PROGRAM WateringTask
VAR
	WaterTimer: TON;
state : INT	 :=0; 	
Delay: Ton;
END_VAR

 	
//Watering control
CASE state OF
	
END_CASE
0:// Initial position
WaterON:= FALSE;
state:=1;
1:// Checking the conditions
IF WaterRequired THEN
            WaterDuration := GetWaterDuration(Moisture, Temp);
            WaterOn := TRUE;
            WaterTimer(IN := TRUE, PT := WaterDuration);
            nState := 2;
        ELSE
            nState := 3;
        END_IF;
		
2:  // Watering
WaterTimer(IN := TRUE);
        IF WaterTimer.Q THEN
          WaterON := FALSE;
WaterRequired := FALSE;
WaterTimer(IN := FALSE);
            state := 3;
3:// Idle
Delay(IN:=TRUE, PT:=T#5S);
IF NOT(Delay.Q) THEN
	RETURN;
END_IF
Delay(In:=FALSE);
state:=1;		
END_CASE

END_PROGRAM

(* stored: Version 1.1.0.1, ProductVersion 3.1.4024.15
   POU WateringTask: Id {b5a1694e-819d-48dc-a239-eb210722768b}, SpecialFunc None *)
